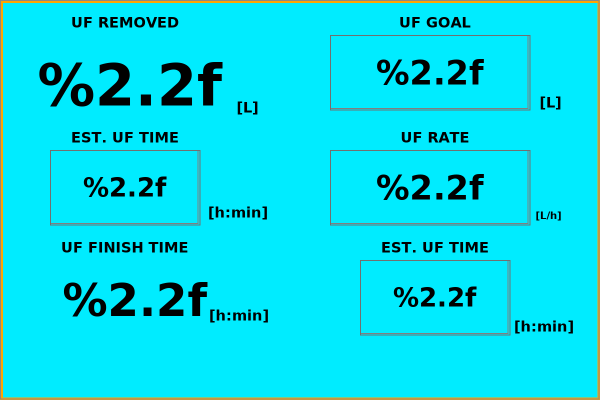
VISUALIZATION RinseMode  // 600x400
    Textfield (0,0 600x400)
    Textfield (50,10 150x25), "UF REMOVED"
    Textfield (360,125 150x25), "UF RATE"
    Textfield (5,35 250x100), "%2.2f"
    Button (330,35 200x75), "%2.2f"
        OnMouseDown: write the text variable via VisuDialogs.Numpad, min 0, max 1000
    Textfield (360,10 150x25), "UF GOAL"
    Button (330,150 200x75), "%2.2f"
        OnMouseDown: write the text variable via VisuDialogs.Numpad, min 0, max 1000
    Button (50,150 150x75), "%2.2f"
        OnMouseDown: write the text variable via VisuDialogs.Numpad, min 0, max 1000
    Textfield (50,125 150x25), "EST. UF TIME"
    Textfield (779,143 1x0)
    Textfield (536,203 25x25), "[L/h]"
    Textfield (538,90 25x25), "[L]"
    Textfield (235,95 25x25), "[L]"
    Textfield (206,200 64x25), "[h:min]"
    Button (360,260 150x75), "%2.2f"
        OnMouseDown: write the text variable via VisuDialogs.Numpad, min 0, max 1000
    Textfield (360,235 150x25), "EST. UF TIME"
    Textfield (512,314 64x25), "[h:min]"
    Textfield (10,250 250x100), "%2.2f"
    Textfield (50,235 150x25), "UF FINISH TIME"
    Textfield (207,303 64x25), "[h:min]"
END_VISUALIZATION

(* stored: Version 1.1.0.1, ProductVersion 3.1.4024.12
   Visu RinseMode: Id {527cf289-e811-4644-848a-a8bf39aff9c0} *)
